// TIA Portal V17 export
// export: Created 2023-12-09T21:24:40.2957917Z, ExportSetting WithDefaults, DisplayName Totally Integrated Automation Portal, DisplayVersion V17, DisplayName TIA Portal Openness, DisplayVersion V17, DisplayName TIA Portal Teamcenter Gateway, DisplayVersion V17, DisplayName TIA Portal Version Control Interface, DisplayVersion V17, DisplayName STEP 7 Professional, DisplayVersion V17, DisplayName STEP 7 Safety, DisplayVersion V17, DisplayName WinCC Advanced / Unified PC, DisplayVersion V17
DATA_BLOCK "dbSend_PLC2fromPLC1"   // DB4
{ S7_Optimized_Access := 'TRUE' }
VERSION : 0.1
// stored: AutoNumber true, IsOnlyStoredInLoadMemory false, IsWriteProtectedInAS false
   VAR
      wyslane : Int;
   END_VAR
BEGIN
END_DATA_BLOCK
